FUNCTION_BLOCK FB_Axis

VAR_INPUT

    //========================================================AXIS SHAPE========================================================
    coilShapeID           : INT := 0;                 // defines shape of coil attached to axis.
    pancake               : pancake_params_0;         // ID 0
    racetrack             : racetrack_params_1;       // ID 1

    //========================================================AXIS DIMENSIONS========================================================
    outerRadiusCurrent    : LREAL :=gvl.MIN_MOUNT_RADIUS/1000; // outer radius of coil

    //========================================================AXIS TAPE========================================================
    tape_info             : POINTER TO ARRAY[0..10] OF tape_info;// array of tape information
    tapeType              : INT;                      // type of tape

    //========================================================MASS========================================================
    emptyMassKG           : LREAL := 20;              // mass of the empty axis in KG
    momentInertia         : LREAL := 0;               // moment of inertia

    //========================================================AXIS CONTROL BOOL========================================================
    // sets which FB's should be executed cyclically
    powerEnable           : BOOL;                     // power enable
    resetEnable           : BOOL;                     // reset enable
    velocityEnable        : BOOL;                     // velocity enable
    haltEnable            : BOOL;                     // halt enable
    homeEnable            : BOOL;                     // home enable
    stopEnable            : BOOL;                     // stop enable
    torqueEnable          : BOOL;                     // torque enable
    posEnable             : BOOL;                     // position enable
    modmoveEnable         : BOOL;                     // move modulo enable
    test                  : BOOL;                     // test enable
    enabled               : BOOL;                     // sets whether axis is enabled
	
    //========================================================AXIS CONTROL MISC OPTIONS========================================================
    // misc options for axis
    directionB            : INT := 0;                 // direction
    direction             : MC_Direction := MC_Positive_Direction; // direction of motion
    buffermode            : MC_BufferMode := MC_Aborting;           // buffer mode
    moveOptions           : ST_MoveOptions;           // move options
    homeOptions           : ST_HomingOptions;         // homing options

    ST_SetPositionOptions : ST_SetPositionOptions;    // set position options

    //========================================================AXIS CONTROL VALUES========================================================
    // TORQUE CONTROL
    torque                : LREAL;                    // torque value
    velocityLimitHigh     : LREAL;                    // high velocity limit
    velocityLimitLow      : LREAL;                    // low velocity limit

    // SECONDARY TORQUE CONTROL SETTINGS
    acceleration          : LREAL := 1800;               // acceleration value
    deceleration          : LREAL := 1800;               // deceleration value
    torqueRamp            : LREAL := 1000;            // torque ramp value

    jerk                  : LREAL := 0;               // jerk value

    // VELOCITY CONTROL
    velocity              : LREAL;                    // velocity value

    //========================================================AXIS STATUS VARS========================================================
    actualTorque          : LREAL;                    // actual torque value
    actualVelocity        : LREAL;                    // actual velocity value
    state                 : INT;                      // state value ((1=powered,2=disabled,3=in motion,4=error))
    adsError              : BOOL;                     // ADS error flag
    adsErrorID            : UDINT;                    // ADS error ID
	errorType			  : UDINT;					  // 1= ads 2= axis 0=no error
	errorID				  : UDINT;					  // error ID, axis errors take precedence over ads errors 	
    //========================================================AXIS PARAMS========================================================
    ratedCurrent          : LREAL;                    // rated current
    torqueConstant        : LREAL;                    // torque constant
    gearRatioNum          : INT;                      // gear ratio numerator
    gearRatioDen          : INT;                      // gear ratio denominator

    //========================================================AXIS CONTROL FB========================================================
    // instantiates FB's for various axis control functions
    MCPOWER               : MC_Power;                 // power control
    MCRESET               : MC_Reset;                 // reset control
    MCHOME                : MC_Home;                  // home control
    MCVELOCITY            : MC_MoveVelocity;          // move velocity control
    MCHALT                : MC_Halt;                  // halt control
    MCSTOP                : MC_Stop;                  // stop control
    MCGETVELOCITY         : MC_ReadActualVelocity;    // read actual velocity
    MCTORQUECONTROL       : MC_TorqueControl;         // torque control
    MCPOS                 : MC_SetPosition;           // set position
    MCJOG                 : MC_Jog;                   // jog control
    MCMOVEMOD             : MC_MoveModulo;            // move modulo control
	MCReadStatus		  : MC_ReadStatus;			  // reads status from motor
	MCWriteParam		  : MC_WriteParameter;
	SoEReset			  : FB_SoEReset;			
    //========================================================AXIS========================================================
    AXIS                  : Axis_REF;                 // axis reference

END_VAR

METHOD CYLIC : BOOL
VAR_INPUT
END_VAR

VAR
	homePosition: LREAL;

	
END_VAR
Axis.ReadStatus();

powerEnable:=enabled; 

MCPOWER(Axis:=Axis,
		Enable:=powerEnable,
		Enable_Positive:=powerEnable,
		Enable_Negative:=powerEnable
		);
		
MCSTOP(Axis:=Axis,
		Execute:=stopEnable,
		Deceleration:=deceleration,
		Jerk:=jerk,Options:=moveOptions);
		
MCHALT(Axis:=Axis,
		Execute:=haltEnable,
		Deceleration:=deceleration,
		Jerk:=jerk,BufferMode:=buffermode,
		Options:=moveOptions);		

	
MCTORQUECONTROL(Axis:=Axis,
				Execute:=torqueEnable,
				ContinuousUpdate:=TRUE,
				Relative:=FALSE,
				Torque:=(torque*100)/(ratedCurrent*torqueConstant),
				TorqueRamp:=torqueRamp,
				VelocityLimitHigh:=velocityLimitHigh,
				VelocityLimitLow:=velocityLimitLow);
				
MCVELOCITY(Axis:=Axis,Execute:=FALSE);

MCVELOCITY(Axis:=Axis,
			Execute:=velocityEnable,
			Acceleration:=acceleration,
			Deceleration:=deceleration,
			Jerk:=jerk,
			Direction:=direction,
			Velocity:=velocity);
			


MCGETVELOCITY(Axis:=AXIS,
			Enable:=TRUE,
			ActualVelocity=>actualVelocity);

	 
getTorque();
stateUpdate();
findinertia();
error_check_all();


errorType:=0; //error type 1 = error inside of a FB. Error type 2 = error op axis. Error type 3= error inside of axis and on axis


IF adserror THEN
	errorType:=errorType +1 ;
	errorID:=adsErrorID;
END_IF
IF axis.Status.Error THEN
	errorType:=errorType +2;
	errorID:=axis.Status.errorid;
END_IF
END_METHOD

METHOD error_check_all : BOOL
VAR_OUTPUT
	
END_VAR

IF(powerEnable) THEN
	power_error_check(Error=>adsError,errorID=>adsErrorID);

END_IF


IF(torqueEnable) THEN
	torque_error_check(Error=>adsError,errorID=>adsErrorID);
END_IF



IF(velocityenable) THEN
	velocity_error_check(Error=>adsError,errorID=>adsErrorID);
END_IF



IF(stopenable) THEN
	stop_error_check(Error=>adsError,errorID=>adsErrorID);
END_IF




IF(posenable) THEN
	setpos_error_check(Error=>adsError,errorID=>adsErrorID);
END_IF
END_METHOD

METHOD findinertia : BOOL
VAR_INPUT
END_VAR

VAR
	cableMassKG: LREAL;
END_VAR
//to do , find mass from cable.

momentInertia:=(0.5)*(emptyMassKG+cableMassKG)*EXPT(getDistToAxis(),2);
END_METHOD

METHOD getDistToAxis : LREAL
VAR_INPUT
END_VAR
//Finds distance to axis from internal dimension and turn count vars. 

//NOTE: this only works for payoff axies. 

//output units in mm. IMPORTANT

CASE coilShapeID OF
	0:
	
	CASE directionB OF
		
	0: //Finds direction if motor is being unwound
	
	getDistToAxis:=(pancake.radius - axis.NcToPlc.ModuloActTurns*tape_info^[tapeType].tape_depth)/1000; 
	
	1: //Finds direction if motor is being wound
	
	getDistToAxis:=(pancake.radius + axis.NcToPlc.ModuloActTurns*tape_info^[tapeType].tape_depth)/1000;
	
	
	END_CASE

END_CASE
END_METHOD

METHOD getTorque : BOOL
VAR_INPUT
END_VAR
actualTorque:=(AXIS.NcToPlc.ActTorque/100)*ratedCurrent*torqueConstant;
//actualTorque:=AXIS.NcToPlc.ActTorque;
END_METHOD

METHOD halt_error_check : BOOL
VAR_INPUT
END_VAR

VAR_OUTPUT
	Error: BOOL;
	errorID: UDINT;
END_VAR
MCHALT(Axis:=Axis,Error=>Error,ErrorID=>errorID);
END_METHOD

METHOD INIT : BOOL
VAR_INPUT
END_VAR

VAR
	i: INT;
END_VAR
powerEnable:=TRUE;

//set options
ST_SetPositionOptions.ClearPositionLag:=TRUE;  

//reset axis to clear any errors
MCRESET(Axis:=AXIS,Execute:=TRUE);
MCRESET(Axis:=AXIS,Execute:=FALSE);
END_METHOD

METHOD power_error_check : BOOL
VAR_OUTPUT
	error :BOOL;
	errorID : UDINT;
END_VAR
MCPOWER(Axis:=Axis,Error=>Error,ErrorID=>errorID);
END_METHOD

METHOD reset : BOOL
VAR_INPUT
END_VAR
MCRESET(Axis:=AXIS,EXECUTE:=FALSE);
MCRESET(Axis:=AXIS,EXECUTE:=TRUE);

errorID:=0;
errorType:=0;
END_METHOD

METHOD setClear : BOOL
VAR_INPUT
END_VAR
velocityEnable:=FALSE;
stopEnable:=FALSE;
haltEnable:=FALSE;
homeEnable:= FALSE;
torqueEnable:= FALSE;
posEnable:=FALSE;
modmoveEnable:=FALSE;
END_METHOD

METHOD setFree : BOOL
VAR_INPUT
END_VAR
velocityEnable:=FALSE;
stopEnable:=FALSE;
haltEnable:=FALSE;
homeEnable:= FALSE;
torqueEnable:= FALSE;
posEnable:=FALSE;
END_METHOD

METHOD setHalt : BOOL
VAR_INPUT
END_VAR
velocityEnable:=FALSE;
stopEnable:=FALSE;
haltEnable:=TRUE;
homeEnable:= FALSE;
torqueEnable:= FALSE;
posEnable:=FALSE;
END_METHOD

METHOD setHome : BOOL
VAR_INPUT
END_VAR
velocityEnable:=FALSE;
stopEnable:=FALSE;
haltEnable:=FALSE;
homeEnable:= TRUE;
torqueEnable:= FALSE;
posEnable:=FALSE;
END_METHOD

METHOD setPos : BOOL
VAR_INPUT
	
END_VAR

VAR
	
	Done: BOOL;
	i: INT;
	busy: BOOL;
END_VAR
END_METHOD

METHOD setpos_error_check : BOOL
VAR_INPUT
END_VAR


VAR_OUTPUT
	Error: BOOL;
	errorID: UDINT;
END_VAR
MCPOS(Axis:=Axis,Error=>Error,ErrorID=>errorID);
END_METHOD

METHOD setReset : BOOL
VAR_INPUT
END_VAR
END_METHOD

METHOD setStop : BOOL
VAR_INPUT
END_VAR
velocityEnable:=FALSE;
stopEnable:=TRUE;
haltEnable:=FALSE;
homeEnable:= FALSE;
torqueEnable:= FALSE;
posEnable:=FALSE;
END_METHOD

METHOD setTorque : BOOL
VAR_INPUT
END_VAR
velocityEnable:=FALSE;
stopEnable:=FALSE;
haltEnable:=FALSE;
homeEnable:= FALSE;
torqueEnable:= TRUE;
posEnable:=FALSE;
END_METHOD

METHOD setVelocity : BOOL
VAR_INPUT
END_VAR
velocityEnable:=TRUE;
stopEnable:=FALSE;
haltEnable:=FALSE;
homeEnable:= FALSE;
torqueEnable:= FALSE;
posEnable:=FALSE;
END_METHOD

METHOD stateUpdate : BOOL
VAR_INPUT
END_VAR
IF powerEnable OR haltEnable OR stopEnable THEN
	state:=1;
END_IF
IF NOT enabled THEN
	state:=2;
END_IF
IF torqueEnable OR velocityEnable OR posEnable THEN
	state:=3;
END_IF
IF AXIS.Status.Error THEN
	state:=4;
END_IF
END_METHOD

METHOD stop_error_check : BOOL
VAR_INPUT
END_VAR

VAR_OUTPUT
	errorID: UDINT;
	Error: BOOL;
END_VAR
MCSTOP(Axis:=Axis,Error=>Error,ErrorID=>errorID);
END_METHOD

METHOD torque_error_check : BOOL
VAR_INPUT
END_VAR

VAR_OUTPUT
	Error: BOOL;
	errorID: UDINT;
END_VAR
MCTORQUECONTROL(Axis:=Axis,Error=>Error,ErrorID=>errorID);
END_METHOD

METHOD velocity_error_check : BOOL
VAR_INPUT
END_VAR

VAR_OUTPUT
	Error: BOOL;
	errorID: UDINT;
END_VAR
MCVELOCITY(Axis:=Axis,Error=>Error,ErrorID=>errorID);
END_METHOD

END_FUNCTION_BLOCK

(* stored: Version 1.1.0.1, ProductVersion 3.1.4024.12
   POU FB_Axis: Id {67c536b7-cb91-42b9-a9d5-7bc5afe11e21}, SpecialFunc None
   Folder Methods: Id {a176b26e-e67a-42bd-94f4-2f0b6113d4b7}
   Folder Error Checks: Id {5e84902a-c5c6-4038-a6b5-6ad92834b0c4}
   Folder Misc: Id {154da71a-12a3-4387-8f76-6b557dc01298}
   Folder sets: Id {31fae47e-262c-4f32-a922-a3f514e3e406}
   Method CYLIC: Id {7c186ae0-44c4-4808-9e23-1f18de41fa53}
   Method error_check_all: Id {d0c59f3f-f6b6-4fd0-853c-e3534ca6d5d0}
   Method findinertia: Id {1c478d19-00ea-4701-b3cf-13a0a384da78}
   Method getDistToAxis: Id {6b2436af-4b54-4ed0-a9cd-4034ab7bf577}
   Method getTorque: Id {6c5c5c23-bebe-4cf8-bf3b-ff120224285b}
   Method halt_error_check: Id {2ca5f59d-5312-4450-b836-ed2e20c6ea56}
   Method INIT: Id {cb6cd0a9-c647-4489-a174-b70a666913ba}
   Method power_error_check: Id {3a006f0e-5221-4ae0-9860-3fc9c0782ddb}
   Method reset: Id {c85d9ad6-d473-4751-8b53-dcece08669b3}
   Method setClear: Id {3edee9ef-4ef0-4a7f-940a-a8847f5820a3}
   Method setFree: Id {d522524d-31a3-418a-824b-ba104553558d}
   Method setHalt: Id {2d8b8748-a52f-4cd2-900f-26056fd38ca1}
   Method setHome: Id {4b055be3-c329-44b4-84a9-fb655fd8c656}
   Method setPos: Id {c270b1b3-4e96-4a7e-92d9-23393108ef68}
   Method setpos_error_check: Id {c1d7af26-a40a-4448-a273-3c6a04d53912}
   Method setReset: Id {704b19ac-a526-4b1d-961a-2b6ba452c168}
   Method setStop: Id {612bcacf-3053-4295-8be1-bb716811093b}
   Method setTorque: Id {37fa63df-8844-4715-be14-1d1e190c6f35}
   Method setVelocity: Id {2e422cbc-a452-44f9-b242-0ddad3731936}
   Method stateUpdate: Id {47b61579-401b-4a3b-b130-c999b128bc7b}
   Method stop_error_check: Id {ef513f0a-80f4-4bef-9122-655fb37b4b98}
   Method torque_error_check: Id {f0391d66-cdcc-462c-8289-6666080e8d59}
   Method velocity_error_check: Id {828667ad-f097-444c-a024-b05a7b520e5b} *)
